# EPICS substitutions: products/ITER/products/org.csstudio.iter.css.product/demo/m-TEST-BOY/src/main/epics/SharedTemplateApp/Db/switch-state.substitutions
file switch-state.db {
    pattern { IOC, COUNT, SCAN }
        { "A", "0", ".1 second" }
        { "A", "1", ".1 second" }
        { "A", "2", ".1 second" }
        { "A", "3", ".1 second" }
        { "A", "4", ".1 second" }
        { "A", "5", ".1 second" }
        { "A", "6", ".1 second" }
        { "A", "7", ".1 second" }
        { "A", "8", ".1 second" }
        { "A", "9", ".1 second" }
        { "A", "10", ".1 second" }
        { "A", "11", ".1 second" }
        { "A", "12", ".1 second" }
        { "A", "13", ".1 second" }
        { "A", "14", ".1 second" }
        { "A", "15", ".1 second" }
        { "A", "16", ".1 second" }
        { "A", "17", ".1 second" }
        { "A", "18", ".1 second" }
        { "A", "19", ".1 second" }
        { "A", "20", ".1 second" }
        { "A", "21", ".1 second" }
        { "A", "22", ".1 second" }
        { "A", "23", ".1 second" }
        { "A", "24", ".1 second" }
        { "A", "25", ".1 second" }
        { "A", "26", ".1 second" }
        { "A", "27", ".1 second" }
        { "A", "28", ".1 second" }
        { "A", "29", ".1 second" }
        { "A", "30", ".1 second" }
        { "A", "31", ".1 second" }
        { "A", "32", ".1 second" }
        { "A", "33", ".1 second" }
        { "A", "34", ".1 second" }
        { "A", "35", ".1 second" }
        { "A", "36", ".1 second" }
        { "A", "37", ".1 second" }
        { "A", "38", ".1 second" }
        { "A", "39", ".1 second" }
        { "A", "40", ".1 second" }
        { "A", "41", ".1 second" }
        { "A", "42", ".1 second" }
        { "A", "43", ".1 second" }
        { "A", "44", ".1 second" }
        { "A", "45", ".1 second" }
        { "A", "46", ".1 second" }
        { "A", "47", ".1 second" }
        { "A", "48", ".1 second" }
        { "A", "49", ".1 second" }
        { "A", "50", ".1 second" }
        { "A", "51", ".1 second" }
        { "A", "52", ".1 second" }
        { "A", "53", ".1 second" }
        { "A", "54", ".1 second" }
        { "A", "55", ".1 second" }
        { "A", "56", ".1 second" }
        { "A", "57", ".1 second" }
        { "A", "58", ".1 second" }
        { "A", "59", ".1 second" }
        { "A", "60", ".1 second" }
        { "A", "61", ".1 second" }
        { "A", "62", ".1 second" }
        { "A", "63", ".1 second" }
        { "A", "64", ".1 second" }
        { "A", "65", ".1 second" }
        { "A", "66", ".1 second" }
        { "A", "67", ".1 second" }
        { "A", "68", ".1 second" }
        { "A", "69", ".1 second" }
        { "A", "70", ".1 second" }
        { "A", "71", ".1 second" }
        { "A", "72", ".1 second" }
        { "A", "73", ".1 second" }
        { "A", "74", ".1 second" }
        { "A", "75", ".1 second" }
        { "A", "76", ".1 second" }
        { "A", "77", ".1 second" }
        { "A", "78", ".1 second" }
        { "A", "79", ".1 second" }
        { "A", "80", ".1 second" }
        { "A", "81", ".1 second" }
        { "A", "82", ".1 second" }
        { "A", "83", ".1 second" }
        { "A", "84", ".1 second" }
        { "A", "85", ".1 second" }
        { "A", "86", ".1 second" }
        { "A", "87", ".1 second" }
        { "A", "88", ".1 second" }
        { "A", "89", ".1 second" }
        { "A", "90", ".1 second" }
        { "A", "91", ".1 second" }
        { "A", "92", ".1 second" }
        { "A", "93", ".1 second" }
        { "A", "94", ".1 second" }
        { "A", "95", ".1 second" }
        { "A", "96", ".1 second" }
        { "A", "97", ".1 second" }
        { "A", "98", ".1 second" }
        { "A", "99", ".1 second" }
        { "A", "100", ".1 second" }
        { "A", "101", ".1 second" }
        { "A", "102", ".1 second" }
        { "A", "103", ".1 second" }
        { "A", "104", ".1 second" }
        { "A", "105", ".1 second" }
        { "A", "106", ".1 second" }
        { "A", "107", ".1 second" }
        { "A", "108", ".1 second" }
        { "A", "109", ".1 second" }
        { "A", "110", ".1 second" }
        { "A", "111", ".1 second" }
        { "A", "112", ".1 second" }
        { "A", "113", ".1 second" }
        { "A", "114", ".1 second" }
        { "A", "115", ".1 second" }
        { "A", "116", ".1 second" }
        { "A", "117", ".1 second" }
        { "A", "118", ".1 second" }
        { "A", "119", ".1 second" }
        { "A", "120", ".1 second" }
        { "A", "121", ".1 second" }
        { "A", "122", ".1 second" }
        { "A", "123", ".1 second" }
        { "A", "124", ".1 second" }
        { "A", "125", ".1 second" }
        { "A", "126", ".1 second" }
        { "A", "127", ".1 second" }
        { "A", "128", ".1 second" }
        { "A", "129", ".1 second" }
        { "A", "130", ".1 second" }
        { "A", "131", ".1 second" }
        { "A", "132", ".1 second" }
        { "A", "133", ".1 second" }
        { "A", "134", ".1 second" }
        { "A", "135", ".1 second" }
        { "A", "136", ".1 second" }
        { "A", "137", ".1 second" }
        { "A", "138", ".1 second" }
        { "A", "139", ".1 second" }
        { "A", "140", ".1 second" }
        { "A", "141", ".1 second" }
        { "A", "142", ".1 second" }
        { "A", "143", ".1 second" }
        { "A", "144", ".1 second" }
        { "A", "145", ".1 second" }
        { "A", "146", ".1 second" }
        { "A", "147", ".1 second" }
        { "A", "148", ".1 second" }
        { "A", "149", ".1 second" }
        { "A", "150", ".1 second" }
        { "A", "151", ".1 second" }
        { "A", "152", ".1 second" }
        { "A", "153", ".1 second" }
        { "A", "154", ".1 second" }
        { "A", "155", ".1 second" }
        { "A", "156", ".1 second" }
        { "A", "157", ".1 second" }
        { "A", "158", ".1 second" }
        { "A", "159", ".1 second" }
        { "A", "160", ".1 second" }
        { "A", "161", ".1 second" }
        { "A", "162", ".1 second" }
        { "A", "163", ".1 second" }
        { "A", "164", ".1 second" }
        { "A", "165", ".1 second" }
        { "A", "166", ".1 second" }
        { "A", "167", ".1 second" }
        { "A", "168", ".1 second" }
        { "A", "169", ".1 second" }
        { "A", "170", ".1 second" }
        { "A", "171", ".1 second" }
        { "A", "172", ".1 second" }
        { "A", "173", ".1 second" }
        { "A", "174", ".1 second" }
        { "A", "175", ".1 second" }
        { "A", "176", ".1 second" }
        { "A", "177", ".1 second" }
        { "A", "178", ".1 second" }
        { "A", "179", ".1 second" }
        { "A", "180", ".1 second" }
        { "A", "181", ".1 second" }
        { "A", "182", ".1 second" }
        { "A", "183", ".1 second" }
        { "A", "184", ".1 second" }
        { "A", "185", ".1 second" }
        { "A", "186", ".1 second" }
        { "A", "187", ".1 second" }
        { "A", "188", ".1 second" }
        { "A", "189", ".1 second" }
        { "A", "190", ".1 second" }
        { "A", "191", ".1 second" }
        { "A", "192", ".1 second" }
        { "A", "193", ".1 second" }
        { "A", "194", ".1 second" }
        { "A", "195", ".1 second" }
        { "A", "196", ".1 second" }
        { "A", "197", ".1 second" }
        { "A", "198", ".1 second" }
        { "A", "199", ".1 second" }
        { "A", "200", ".1 second" }
        { "A", "201", ".1 second" }
        { "A", "202", ".1 second" }
        { "A", "203", ".1 second" }
        { "A", "204", ".1 second" }
        { "A", "205", ".1 second" }
        { "A", "206", ".1 second" }
        { "A", "207", ".1 second" }
        { "A", "208", ".1 second" }
        { "A", "209", ".1 second" }
        { "A", "210", ".1 second" }
        { "A", "211", ".1 second" }
        { "A", "212", ".1 second" }
        { "A", "213", ".1 second" }
        { "A", "214", ".1 second" }
        { "A", "215", ".1 second" }
        { "A", "216", ".1 second" }
        { "A", "217", ".1 second" }
        { "A", "218", ".1 second" }
        { "A", "219", ".1 second" }
        { "A", "220", ".1 second" }
        { "A", "221", ".1 second" }
        { "A", "222", ".1 second" }
        { "A", "223", ".1 second" }
        { "A", "224", ".1 second" }
        { "A", "225", ".1 second" }
        { "A", "226", ".1 second" }
        { "A", "227", ".1 second" }
        { "A", "228", ".1 second" }
        { "A", "229", ".1 second" }
        { "A", "230", ".1 second" }
        { "A", "231", ".1 second" }
        { "A", "232", ".1 second" }
        { "A", "233", ".1 second" }
        { "A", "234", ".1 second" }
        { "A", "235", ".1 second" }
        { "A", "236", ".1 second" }
        { "A", "237", ".1 second" }
        { "A", "238", ".1 second" }
        { "A", "239", ".1 second" }
        { "A", "240", ".1 second" }
        { "A", "241", ".1 second" }
        { "A", "242", ".1 second" }
        { "A", "243", ".1 second" }
        { "A", "244", ".1 second" }
        { "A", "245", ".1 second" }
        { "A", "246", ".1 second" }
        { "A", "247", ".1 second" }
        { "A", "248", ".1 second" }
        { "A", "249", ".1 second" }
        { "A", "250", ".1 second" }
        { "A", "251", ".1 second" }
        { "A", "252", ".1 second" }
        { "A", "253", ".1 second" }
        { "A", "254", ".1 second" }
        { "A", "255", ".1 second" }
        { "A", "256", ".1 second" }
        { "A", "257", ".1 second" }
        { "A", "258", ".1 second" }
        { "A", "259", ".1 second" }
}
